TYPE "PLC_TO_KISTLER"
VERSION : 0.1
   STRUCT
      "0.0" : Bool;
      "0.1" : Bool;
      "0.2" : Bool;
      "0.3" : Bool;
      "0.4" : Bool;
      "0.5" : Bool;
      "0.6" : Bool;
      "0.7" : Bool;
      "1.0" : Bool;
      "1.1" : Bool;
      "1.2" : Bool;
      "1.3" : Bool;
      "1.4" : Bool;
      "1.5" : Bool;
      "1.6" : Bool;
      "1.7" : Bool;
      "2" : Byte;
      "3.0" : Bool;
      "3.1" : Bool;
      "3.2" : Bool;
      "3.3" : Bool;
      "3.4" : Bool;
      "3.5" : Bool;
      "3.6" : Bool;
      "3.7" : Bool;
      "4.0" : Bool;
      "4.1" : Bool;
      "4.2" : Bool;
      "4.3" : Bool;
      "4.4" : Bool;
      "4.5" : Bool;
      "4.6" : Bool;
      "4.7" : Bool;
      "5.0" : Bool;
      "5.1" : Bool;
      "5.2" : Bool;
      "5.3" : Bool;
      "5.4" : Bool;
      "5.5" : Bool;
      "5.6" : Bool;
      "5.7" : Bool;
      "6.0" : Bool;
      "6.1" : Bool;
      "6.2" : Bool;
      "6.3" : Bool;
      "6.4" : Bool;
      "6.5" : Bool;
      "6.6" : Bool;
      "6.7" : Bool;
      "7.0" : Bool;
      "7.1" : Bool;
      "7.2" : Bool;
      "7.3" : Bool;
      "7.4" : Bool;
      "7.5" : Bool;
      "7.6" : Bool;
      "7.7" : Bool;
      "8.0" : Bool;
      "8.1" : Bool;
      "8.2" : Bool;
      "8.3" : Bool;
      "8.4" : Bool;
      "8.5" : Bool;
      "8.6" : Bool;
      "8.7" : Bool;
      "9.0" : Bool;
      "9.1" : Bool;
      "9.2" : Bool;
      "9.3" : Bool;
      "9.4" : Bool;
      "9.5" : Bool;
      "9.6" : Bool;
      "9.7" : Bool;
      "10.0" : Bool;
      "10.1" : Bool;
      "10.2" : Bool;
      "10.3" : Bool;
      "10.4" : Bool;
      "10.5" : Bool;
      "10.6" : Bool;
      "10.7" : Bool;
      "11" : Byte;
      "12" : Byte;
      "13" : Byte;
      "14" : Byte;
      "15.0" : Bool;
      "15.1" : Bool;
      "15.2" : Bool;
      "15.3" : Bool;
      "15.4" : Bool;
      "15.5" : Bool;
      "15.6" : Bool;
      "15.7" : Bool;
      "16" : Byte;
      "17" : Byte;
      "18.0" : Bool;
      "18.1" : Bool;
      "18.2" : Bool;
      "18.3" : Bool;
      "18.4" : Bool;
      "18.5" : Bool;
      "18.6" : Bool;
      "18.7" : Bool;
      "19.0" : Bool;
      "19.1" : Bool;
      "19.2" : Bool;
      "19.3" : Bool;
      "19.4" : Bool;
      "19.5" : Bool;
      "19.6" : Bool;
      "19.7" : Bool;
      "20" : Array[1..50] of Char;
      "70" : Real;
      "74" : Real;
      EO_01 : Struct
         X_Position_LL : Real;
         X_Position_UL : Real;
         Y_Force_LL : Real;
         Y_Force_UL : Real;
      END_STRUCT;
      EO_02 : Struct
         X_Position_LL : Real;
         X_Position_UL : Real;
         Y_Force_LL : Real;
         Y_Force_UL : Real;
      END_STRUCT;
      EO_03 : Struct
         X_Position_LL : Real;
         X_Position_UL : Real;
         Y_Force_LL : Real;
         Y_Force_UL : Real;
      END_STRUCT;
      EO_04 : Struct
         X_Position_LL : Real;
         X_Position_UL : Real;
         Y_Force_LL : Real;
         Y_Force_UL : Real;
      END_STRUCT;
      EO_05 : Struct
         X_Position_LL : Real;
         X_Position_UL : Real;
         Y_Force_LL : Real;
         Y_Force_UL : Real;
      END_STRUCT;
      EO_06 : Struct
         X_Position_LL : Real;
         X_Position_UL : Real;
         Y_Force_LL : Real;
         Y_Force_UL : Real;
      END_STRUCT;
      "174" : Array[1..46] of Byte;
   END_STRUCT;

END_TYPE

